FUNCTION_BLOCK EM_Stamp IMPLEMENTS  ITF_EM_Stamp
VAR_INPUT
END_VAR
VAR_OUTPUT
END_VAR
VAR
END_VAR

END_FUNCTION_BLOCK

(* stored: Version 1.1.0.1, ProductVersion 3.1.4024.12
   POU EM_Stamp: Id {0e46a50c-be27-4c21-a0c4-129444272450}, SpecialFunc None *)
